// TIA Portal V20 export
VAR_GLOBAL   // PLC tag table "Variables Globales Base"
   "FP_0_1 seg" AT %M2.0 : Bool;
   "FP_0_2 seg" AT %M2.1 : Bool;
   "FP_0_4 seg" AT %M2.2 : Bool;
   "FP_0_5 seg" AT %M2.3 : Bool;
   "FP_0_8 seg" AT %M2.4 : Bool;
   "FP_1 seg" AT %M2.5 : Bool;
   "FP_1_6 seg" AT %M2.6 : Bool;
   "FP_2 seg" AT %M2.7 : Bool;
   OFF AT %M10.2 : Bool;
   ON AT %M10.1 : Bool;
   "MAux_1 seg" AT %M1.5 : Bool;
   "MAux_1_6 seg" AT %M1.6 : Bool;
   "MAux_2 seg" AT %M1.7 : Bool;
   "0_1 seg" AT %M0.0 : Bool;   //    {ExternalAccessible false}
   "0_2 seg" AT %M0.1 : Bool;
   "0_4 seg" AT %M0.2 : Bool;
   "0_5 seg" AT %M0.3 : Bool;
   "0_8 seg" AT %M0.4 : Bool;
   "1 seg" AT %M0.5 : Bool;
   "1_6 seg" AT %M0.6 : Bool;
   "2 seg" AT %M0.7 : Bool;
   Rst_Comm_Pantalla_03 AT %T13 : Timer;
   Rst_Comm_Pantalla_02 AT %T12 : Timer;
   Rst_Comm_Pantalla_01 AT %T11 : Timer;
   Rst_Comm_Pantalla_10 AT %T20 : Timer;
   Rst_Comm_Pantalla_09 AT %T19 : Timer;
   Rst_Comm_Pantalla_08 AT %T18 : Timer;
   Rst_Comm_Pantalla_07 AT %T17 : Timer;
   Rst_Comm_Pantalla_06 AT %T16 : Timer;
   Rst_Comm_Pantalla_05 AT %T15 : Timer;
   Rst_Comm_Pantalla_04 AT %T14 : Timer;
   Activar_Simulador AT %M7.0 : Bool;
   Activar_JDT01 AT %M7.1 : Bool;
   Activar_CCPIF_A AT %M3.0 : Bool;
   Activar_CCPIF_B AT %M3.1 : Bool;
   TMP_Pantalla_01 AT %T1 : Timer;
   TMP_Pantalla_10 AT %T10 : Timer;
   TMP_Pantalla_09 AT %T9 : Timer;
   TMP_Pantalla_08 AT %T8 : Timer;
   TMP_Pantalla_07 AT %T7 : Timer;
   TMP_Pantalla_06 AT %T6 : Timer;
   TMP_Pantalla_05 AT %T5 : Timer;
   TMP_Pantalla_04 AT %T4 : Timer;
   TMP_Pantalla_03 AT %T3 : Timer;
   TMP_Pantalla_02 AT %T2 : Timer;
   TMP_Pantalla AT %T0 : Timer;
   AuxTemp_Display AT %M10.0 : Bool;
   AuxTemp_ValorDisplay AT %MD12 : UDInt;
   "MAux_0_1 seg" AT %M1.0 : Bool;
   "MAux_0_2 seg" AT %M1.1 : Bool;
   "MAux_0_4 seg" AT %M1.2 : Bool;
   "MAux_0_5 seg" AT %M1.3 : Bool;
   "MAux_0_8 seg" AT %M1.4 : Bool;
   Error_Display AT %MW20 : UInt;
   Tipo_Display AT %MW16 : UInt;
   Numero_Display AT %MW18 : UInt;
   Activar_JDT02 AT %M7.2 : Bool;
   Activar_CambiarUTDesdeJDT AT %M7.3 : Bool;
   Activar_CCPIF_C AT %M3.2 : Bool;
   TMP_TPDW_OK AT %M20.0 : Bool;
   TMP_TP2DW_OK AT %M20.1 : Bool;
   TMP_TPDW_E1S3_OK AT %M22.0 : Bool;
   TMP_TPDW_E2S4_OK AT %M22.1 : Bool;
   TMP_TRDW_OK AT %M22.2 : Bool;
   Activar_JdTAntiguo AT %M7.4 : Bool;
   Memo_JdTAntiguo_Desactivado AT %M7.5 : Bool;
   Memo_JdTAntiguo_Activado AT %M7.6 : Bool;
END_VAR
VAR_GLOBAL CONSTANT   // user constants
   CTE_MaxMesas : UInt := 500;   // Maximo numero de Mesas de la Instalacion
   CTE_MaxUTs : UInt := 1000;   // Maximo numero de UT's de la Instalacion
   CTE_MaxDispositivos : UInt := 100;   // Maximo numero de Dispositivos CBOX (El CCPIF es 0)
   CTE_TMPEsperaFinReset : UDInt := 60;   // Tiempo de Espera de Fin de Reset (60 Segundos)
   CTE_TMPEsperaFinParoBlando : UDInt := 60;   // Tiempo de Espera de Fin de Paro Blando (60 Segundos)
   CTE_BaseUnidades_100ms : UDInt := 100;
   CTE_BaseUnidades_1ms : UDInt := 1;
   CTE_OffsetCCPIF : UInt := 0;   // Cuanto se suma para saber el Numero de CCPIF del MFS (JdT)
   CTE_OffsetMesa : UInt := 1000;   // Cuanto se suma para saber el Numero de Mesa del MFS (JdT)
   CTE_MaxTodosDispositivos : UInt := 1200;   // ( MaxMesas+MaxDispositivos ) * 2
   CTE_MaxDispositivosBaliza : UInt := 500;   // Maximo Numero de Dispositivos Baliza
   CTE_MaxDispositivosLlave : UInt := 500;   // Maximo Numero de Dispositivos Llave
   CTE_MaxDispositivosSeta : UInt := 500;   // Maximo Numero de Dispositivos Seta
   CTE_MaxDispositivosBarrera : UInt := 500;   // Maximo Numero de Dispositivos Barrera
   CTE_MaxDispositivosPuerta : UInt := 500;   // Maximo Numero de Dispositivos Puerta
   CTE_MaxDispositivosLineaPotencia : UInt := 500;   // Maximo Numero de Dispositivos Linea de Potencia
   V_TMP_EsperaEnTension : Int := 3000;   // Tiempo en Espera En Tension de la Mesa
   CTE_BaseUnidades_1s : UDInt := 1000;
   CTE_FiltroTRElectrico : Int := 200;   // Filtro Error TR Electrico
END_VAR
